(* CODESYS project bo_epc_io001_example_project.project
   Title: BO_EPC_IO001 Example Project
   Version: 1.0.0.0
   Company: Janz Tec AG

Project tree, tasks and I/O mapping:
  Device : Janz emCONTROL Dynamic 64Bit, Janz Tec AG, version 3.5.14.20
    application Application
      libraries: Standard, * (System)
      task MainTask (cyclic, interval 4 ms, priority 1) calls PLC_PRG
      task VISU_TASK (cyclic, interval 100 ms, priority 31) calls VisuElems.Visu_Prg
      program PLC_PRG [ST]
      visualisation Visualization
      visualisation AnalogVisu
    SoftMotion General Axis Pool
    BO_EPC_IO001 : BO_EPC_IO001, Janz Tec AG, version 3.5.11.0
        input  Application.PLC_PRG.digitalinputs : BYTE  // digital inputs
        input  Application.PLC_PRG.analoginputs[0] : REAL  // analog input 1
        input  Application.PLC_PRG.analoginputs[1] : REAL  // analog input 2
        input  Application.PLC_PRG.analoginputs[2] : REAL  // analog input 3
        input  Application.PLC_PRG.analoginputs[3] : REAL  // analog input 4
        output Application.PLC_PRG.digitaloutputs : BYTE  // digital outputs
        output Application.PLC_PRG.analogoutputs[0] : REAL  // analog output 1
        output Application.PLC_PRG.analogoutputs[1] : REAL  // analog output 2
        output Application.PLC_PRG.analogoutputs[2] : REAL  // analog output 3
        output Application.PLC_PRG.analogoutputs[3] : REAL  // analog output 4
        unmapped channels: error code
  text list GlobalTextList
*)

// Device/Application/PLC_PRG
PROGRAM PLC_PRG
VAR
	digitalinputs : BYTE;
	digitaloutputs : BYTE;
	analoginputs :ARRAY[0..3] OF REAL; // -10V..10V
	analogoutputs :ARRAY[0..3] OF REAL; // -10V..10V
	
	 

END_VAR

;

END_PROGRAM

// Device/Application/Visualization
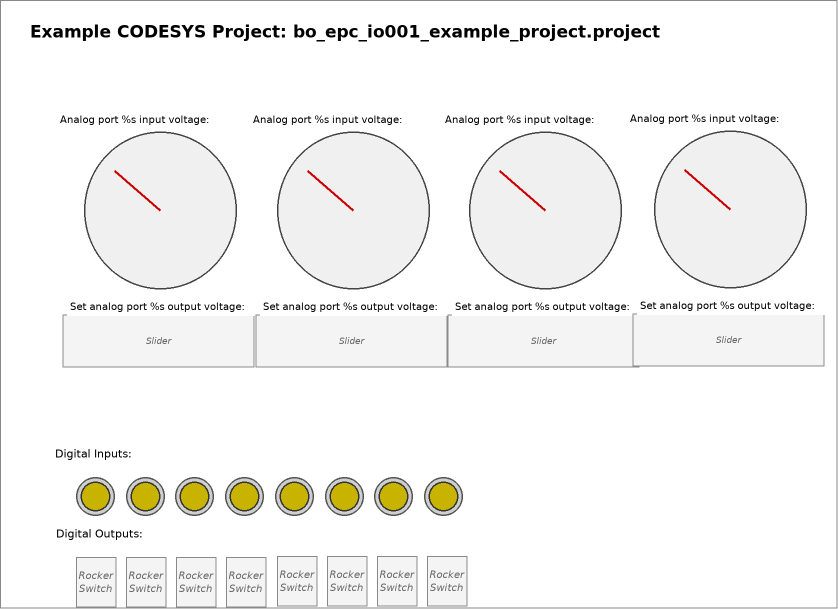
VISUALIZATION Visualization  // 838x609
    Frame (31,107 235x262)
        shows AnalogVisu(index := 0)
    Frame (224,107 235x262)
        shows AnalogVisu(index := 1)
    Frame (416,107 235x262)
        shows AnalogVisu(index := 2)
    Frame (601,106 235x262)
        shows AnalogVisu(index := 3)
    Lamp1 (73,473 45x47), variable: PLC_PRG.digitalinputs.0, style: Lamp-Lamp1-Yellow
    Lamp1 (123,473 45x47), variable: PLC_PRG.digitalinputs.1, style: Lamp-Lamp1-Yellow
    Lamp1 (172,473 45x47), variable: PLC_PRG.digitalinputs.2, style: Lamp-Lamp1-Yellow
    Lamp1 (222,473 45x47), variable: PLC_PRG.digitalinputs.3, style: Lamp-Lamp1-Yellow
    Lamp1 (272,473 45x47), variable: PLC_PRG.digitalinputs.4, style: Lamp-Lamp1-Yellow
    Lamp1 (322,473 45x47), variable: PLC_PRG.digitalinputs.5, style: Lamp-Lamp1-Yellow
    Lamp1 (371,473 45x47), variable: PLC_PRG.digitalinputs.6, style: Lamp-Lamp1-Yellow
    Lamp1 (421,473 45x47), variable: PLC_PRG.digitalinputs.7, style: Lamp-Lamp1-Yellow
    Rectangle (52,444 222x20), "Digital Inputs:"
    Rectangle (53,524 222x20), "Digital Outputs:"
    RockerSwitch (76,557 40x50), variable: PLC_PRG.digitaloutputs.0, behaviour: TOGGLE, style: Switch-RockerSwitch-Gray
    RockerSwitch (126,557 40x50), variable: PLC_PRG.digitaloutputs.1, behaviour: TOGGLE, style: Switch-RockerSwitch-Gray
    RockerSwitch (176,557 40x50), variable: PLC_PRG.digitaloutputs.2, behaviour: TOGGLE, style: Switch-RockerSwitch-Gray
    RockerSwitch (226,557 40x50), variable: PLC_PRG.digitaloutputs.3, behaviour: TOGGLE, style: Switch-RockerSwitch-Gray
    RockerSwitch (277,556 40x50), variable: PLC_PRG.digitaloutputs.4, behaviour: TOGGLE, style: Switch-RockerSwitch-Gray
    RockerSwitch (327,556 40x50), variable: PLC_PRG.digitaloutputs.5, behaviour: TOGGLE, style: Switch-RockerSwitch-Gray
    RockerSwitch (377,556 40x50), variable: PLC_PRG.digitaloutputs.6, behaviour: TOGGLE, style: Switch-RockerSwitch-Gray
    RockerSwitch (427,556 40x50), variable: PLC_PRG.digitaloutputs.7, behaviour: TOGGLE, style: Switch-RockerSwitch-Gray
    Rectangle (27,16 713x31), "Example CODESYS Project: bo_epc_io001_example_project.project"
END_VISUALIZATION

// Device/Application/AnalogVisu
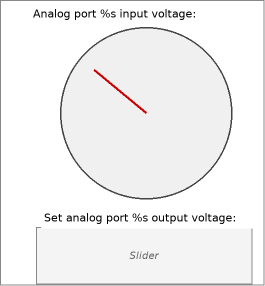
VISUALIZATION AnalogVisu  // 265x286
VAR_INPUT
	index: INT;
END_VAR
    Meter360 (56,27 180x172), value: PLC_PRG.analoginputs[index], style: Meter-Meter360-Gray, scale format: %.1f, scale -10..10
        p518627256: [V]
    Slider (36,227 216x57), variable: PLC_PRG.analogoutputs[index], scale -10..10
    Rectangle (30,4 222x20), "Analog port %s input voltage:", text variable: index
    Rectangle (41,208 222x20), "Set analog port %s output voltage:", text variable: index
END_VISUALIZATION
